{attribute 'OPC.UA.DA' := '0'}
TYPE HTPowermeter :
STRUCT
	PolarisationConfig : PolarisationConfig;
	RFactorSettings : RFactorSettings;
	ResponsivityConfig : ResponsivityConfig;
END_STRUCT
END_TYPE

(* stored: Version 1.1.0.1, ProductVersion 3.1.4024.10
   DUT HTPowermeter: Id {0872520f-b9b5-43c3-90f8-280a9e4f1c94} *)
